Fanuc KAREL source: POP_KEY_RD.kl

PROGRAM T
%NOLOCKGROUP
VAR
 v0 : STRING[40]
 v1 : INTEGER
 v2 : INTEGER
BEGIN
 POP_KEY_RD(v0, v1, v2)
END T
